# B&R Automation Studio project Lab1_pomrs
Automation Studio 4.5.2.102


## Logical view

Binary libraries used (declarations not repeated): operator, runtime, astime, AsIecCon

### Library Logical/Libraries/Library_MC (ANSIC)

#### Library_MC.fun - Exported functions and function blocks
```iecst
{REDUND_ERROR} FUNCTION_BLOCK FB_Motor (*TODO: Add your comment here*) (*$GROUP=User,$CAT=User,$GROUPICON=User.png,$CATICON=User.png*)
	VAR_INPUT
		u : {REDUND_UNREPLICABLE} REAL;
	END_VAR
	VAR_OUTPUT
		w : REAL;
		phi : REAL;
	END_VAR
	VAR
		integrator : FB_Integrator;
		Tm : REAL;
		ke : REAL;
		dt : REAL;
	END_VAR
END_FUNCTION_BLOCK

{REDUND_ERROR} FUNCTION_BLOCK FB_Regulator (*TODO: Add your comment here*) (*$GROUP=User,$CAT=User,$GROUPICON=User.png,$CATICON=User.png*)
	VAR_INPUT
		e : {REDUND_UNREPLICABLE} REAL;
	END_VAR
	VAR_OUTPUT
		u : REAL;
	END_VAR
	VAR
		k_p : REAL;
		k_i : REAL;
		integrator : FB_Integrator;
		iyOld : REAL;
		max_abs_value : REAL;
		dt : REAL;
	END_VAR
END_FUNCTION_BLOCK

{REDUND_ERROR} {REDUND_UNREPLICABLE} FUNCTION_BLOCK FB_Integrator (*TODO: Add your comment here*) (*$GROUP=User,$CAT=User,$GROUPICON=User.png,$CATICON=User.png*)
	VAR_INPUT
		in : {REDUND_UNREPLICABLE} REAL;
	END_VAR
	VAR_OUTPUT
		out : {REDUND_UNREPLICABLE} REAL;
	END_VAR
	VAR
		dt : {REDUND_UNREPLICABLE} REAL;
	END_VAR
END_FUNCTION_BLOCK
```

#### FB_Motor.c
```c
#include <bur/plctypes.h>
#ifdef __cplusplus
	extern "C"
	{
#endif
	#include "Library_MC.h"
#ifdef __cplusplus
	};
#endif
/* TODO: Add your comment here */
void FB_Motor(struct FB_Motor* inst)
{

	/*TODO: Add your code here*/

	inst->w   = (inst->u*(1/inst->ke)-inst->w)*(1/inst->Tm);

	inst->integrator.in = inst->w;
	FB_Integrator(&inst->integrator);
	inst->w=inst->integrator.out;

	inst->integrator.in = inst->w;
	FB_Integrator(&inst->integrator);
	inst->phi = inst->integrator.out;
}
```

#### FB_Regulator.c
```c
#include <bur/plctypes.h>
#ifdef __cplusplus
	extern "C"
	{
#endif
	#include "Library_MC.h"
#ifdef __cplusplus
	};
#endif
/* TODO: Add your comment here */
void FB_Regulator(struct FB_Regulator* inst)
{
	REAL u1;
	REAL u2;
	REAL sum_u;
	/*TODO: Add your code here*/
	u1 = inst->e*inst->k_p;

	if ((u1)>inst->max_abs_value || u1<-inst->max_abs_value)
	{
		if (u1>0)
		{
			u1 = inst->max_abs_value;
		}
		if (u1<0)
		{
			u1 = -inst->max_abs_value;
		}
	}

	u2 = inst->e*inst->k_i + inst->iyOld;

	inst->integrator.in = u2;
	FB_Integrator(&(inst->integrator));
	u2=inst->integrator.out;

	sum_u = u1+u2;

	if (sum_u>inst->max_abs_value || sum_u<-inst->max_abs_value)
	{
		if (sum_u>0)
		{
			sum_u = inst->max_abs_value;
		}
		if (sum_u<0)
		{
			sum_u = -inst->max_abs_value;
		}
	}
	inst->u = sum_u;
	inst->iyOld = inst->u - sum_u;

}
```

#### FB_Integrator.c
```c
#include <bur/plctypes.h>
#ifdef __cplusplus
	extern "C"
	{
#endif
	#include "Library_MC.h"
#ifdef __cplusplus
	};
#endif
/* TODO: Add your comment here */
void FB_Integrator(struct FB_Integrator* inst)
{
	/*TODO: Add your code here*/
	inst->dt=0.02;
	inst->out = inst->dt*inst->in + inst->out;

}
```

### Program Logical/Program

#### Variables.var
```iecst
VAR
	fb_regulator : FB_Regulator;
	fb_motor : FB_Motor;
	Enable : BOOL := FALSE;
	Speed : REAL := 0;
	e : REAL := 0;
	exit_speed : REAL := 0;
	cnt : REAL := 0.0;
	fb_motor_unreg : FB_Motor;
	exit_speed_unreg : REAL;
	u_unreg : REAL := 0.0;
	pulse_width : REAL := 0;
END_VAR
```

#### Cyclic.c
```c
#include <bur/plctypes.h>

#ifdef _DEFAULT_INCLUDES
	#include <AsDefault.h>
#endif

void _CYCLIC ProgramCyclic(void)
{

	//Speed = 10;
	if (Enable)
	{
		cnt += 1;
		if (cnt >= 10 && cnt <= pulse_width)
		{
			Speed = 5;
		}
		else
		{
			Speed = 0;
		//	u_unreg = 0;
		}

		e = Speed*3.14/30 - fb_motor.w;
		fb_regulator.e = e;
		FB_Regulator(&fb_regulator);
		fb_motor.u = fb_regulator.u * fb_motor.ke;
		fb_motor_unreg.u = Speed*3.14/30*fb_motor.ke;
		FB_Motor(&fb_motor_unreg);
		FB_Motor(&fb_motor);
		exit_speed = fb_motor.w*(30/3.14);
		exit_speed_unreg = fb_motor_unreg.w*(30/3.14);
	}
	else
	{
		cnt = 0;
	}
}
```

#### Init.c
```c
#include <bur/plctypes.h>

#ifdef _DEFAULT_INCLUDES
	#include <AsDefault.h>
#endif

void _INIT ProgramInit(void)
{
	Enable = 0;
	Speed = 0;
	pulse_width = 50;

	fb_motor.dt=0.02;
	fb_motor.ke=43.3;
	fb_motor.Tm=0.17;

	fb_motor_unreg.dt = 0.02;
	fb_motor_unreg.ke=43.3;
	fb_motor_unreg.Tm=0.17;

	fb_regulator.dt = 0.02;
	fb_regulator.k_p = 7.361;//3.804;
	fb_regulator.k_i =43.3;
	fb_regulator.max_abs_value = 24;

}
```

Listed in the project but not available here: Logical/Libraries/Library_MC/Types.typ, Logical/Libraries/Library_MC/Constants.var
